FUNCTION_BLOCK fbMotorInverterCtrl

VAR_INPUT
	IN_DevName:STRING;
	In_Enable:BOOL;
	In_Reset:BOOL;

	(*Inverter Healthy Signal*)
	In_InvRdy:BOOL;

END_VAR

VAR_OUTPUT
	Out_InvRun:BOOL;
	Out_InvDirc:BOOL;
	Out_InvSpdBit0:BOOL;
	Out_InvSpdBit1:BOOL;

END_VAR

VAR_IN_OUT
	MotorVar:structMotorInverter;	
	Station:structStationCtrl;
END_VAR


VAR

	MotorOn:BOOL;
	On_TOut: TON;
	On_TON: TON;
	NotRdy_TON:	TON;
	Loc_OnPls: BOOL;
	OnPls: R_TRIG;
	Out_RSErr:BOOL;
	OnPosPls: F_TRIG;
	TempInt:INT;

	pls_ManualModeOff: R_trig;
END_VAR

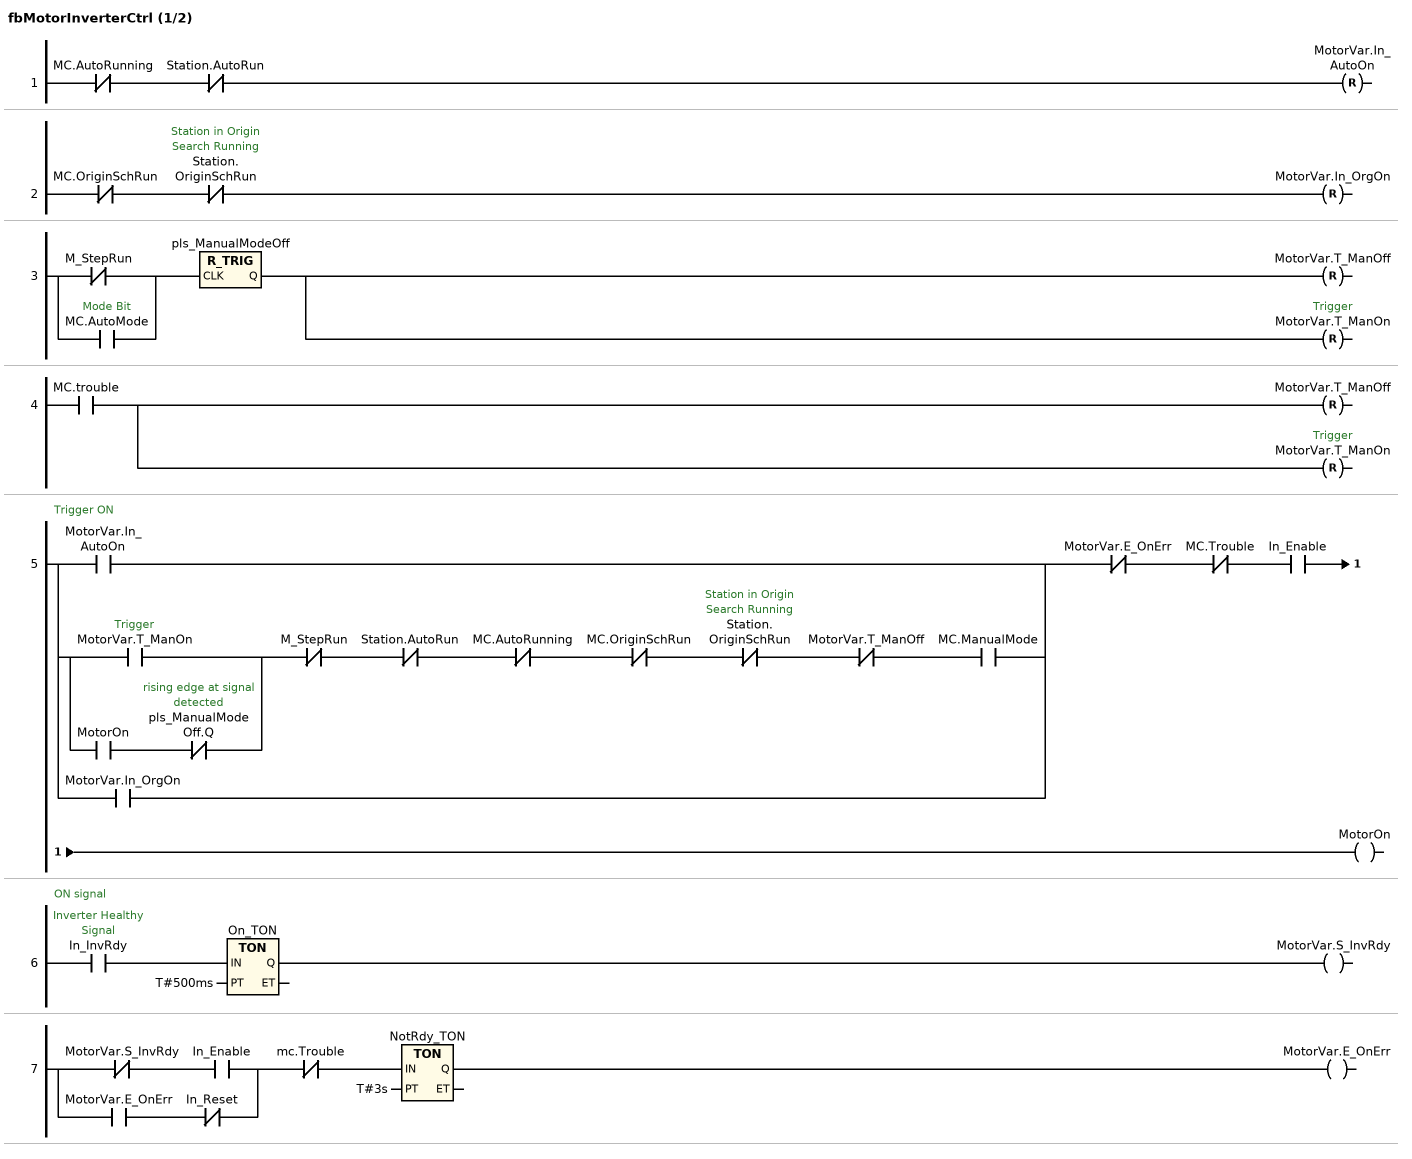
// NETWORK 1
MotorVar.In_AutoOn R= NOT MC.AutoRunning AND NOT Station.AutoRun;

// NETWORK 2
//   Station.OriginSchRun: Station in Origin Search Running
MotorVar.In_OrgOn R= NOT MC.OriginSchRun AND NOT Station.OriginSchRun;

// NETWORK 3
//   MC.AutoMode: Mode Bit
//   MotorVar.T_ManOn: Trigger
pls_ManualModeOff(CLK := NOT M_StepRun OR MC.AutoMode); // R_TRIG
MotorVar.T_ManOff R= pls_ManualModeOff.Q;
MotorVar.T_ManOn R= pls_ManualModeOff.Q;

// NETWORK 4
//   MotorVar.T_ManOn: Trigger
MotorVar.T_ManOff R= MC.trouble;
MotorVar.T_ManOn R= MC.trouble;

// NETWORK 5
// Trigger ON
//   MotorVar.T_ManOn: Trigger
//   pls_ManualModeOff.Q: rising edge at signal detected
//   Station.OriginSchRun: Station in Origin Search Running
MotorOn := (MotorVar.In_AutoOn OR (MotorVar.T_ManOn OR MotorOn AND NOT pls_ManualModeOff.Q) AND NOT M_StepRun AND NOT Station.AutoRun AND NOT MC.AutoRunning AND NOT MC.OriginSchRun AND NOT Station.OriginSchRun AND NOT MotorVar.T_ManOff AND MC.ManualMode OR MotorVar.In_OrgOn) AND NOT MotorVar.E_OnErr AND NOT MC.Trouble AND In_Enable;

// NETWORK 6
// ON signal
//   In_InvRdy: Inverter Healthy Signal
On_TON(IN := In_InvRdy, PT := T#500ms); // TON
MotorVar.S_InvRdy := On_TON.Q;

// NETWORK 7
NotRdy_TON(IN := (NOT MotorVar.S_InvRdy AND In_Enable OR MotorVar.E_OnErr AND NOT In_Reset) AND NOT mc.Trouble, PT := T#3s); // TON
MotorVar.E_OnErr := NotRdy_TON.Q;

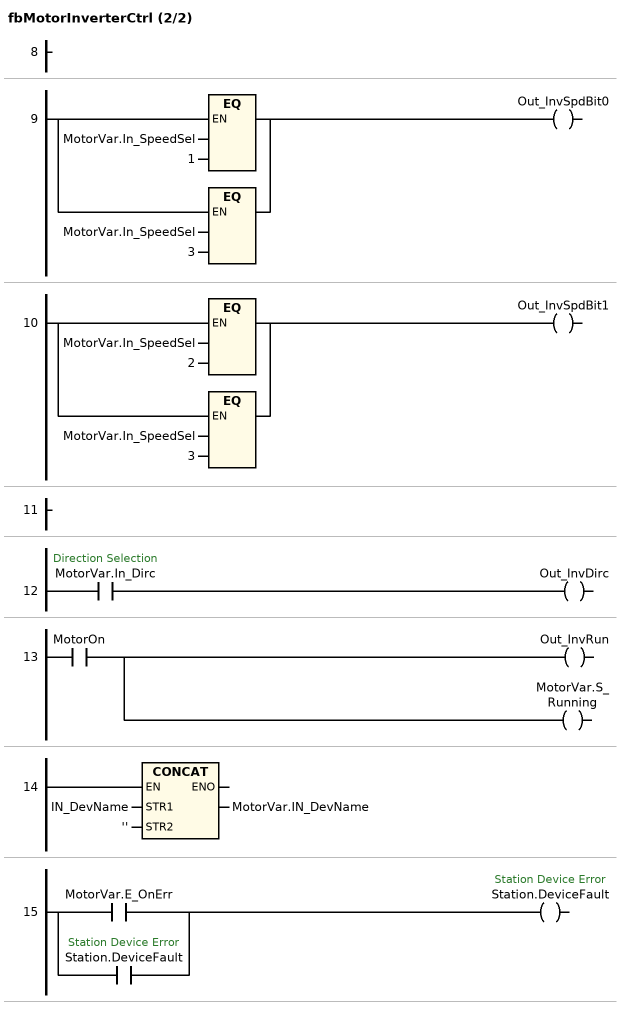
// NETWORK 8

// NETWORK 9
//   MotorVar.In_SpeedSel: Speed Selection 0-3
Out_InvSpdBit0 := MotorVar.In_SpeedSel = 1 OR MotorVar.In_SpeedSel = 3;

// NETWORK 10
//   MotorVar.In_SpeedSel: Speed Selection 0-3
Out_InvSpdBit1 := MotorVar.In_SpeedSel = 2 OR MotorVar.In_SpeedSel = 3;

// NETWORK 11

// NETWORK 12
//   MotorVar.In_Dirc: Direction Selection
Out_InvDirc := MotorVar.In_Dirc;

// NETWORK 13
Out_InvRun := MotorOn;
MotorVar.S_Running := MotorOn;

// NETWORK 14
MotorVar.IN_DevName := CONCAT(STR1 := IN_DevName, STR2 := '');

// NETWORK 15
//   Station.DeviceFault: Station Device Error
Station.DeviceFault := MotorVar.E_OnErr OR Station.DeviceFault;

END_FUNCTION_BLOCK

(* stored: Version 1.1.0.1, ProductVersion 3.1.4018.2
   POU fbMotorInverterCtrl: Id {adce049c-7112-4a9d-b6ad-8836b7b4a95c}, SpecialFunc None *)
